Fanuc TP program (LS listing): DOOR_NOT_OP.LS

/PROG  DOOR_NOT_OP
/ATTR
OWNER		= MNEDITOR;
COMMENT		= "";
PROG_SIZE	= 170;
CREATE		= DATE 25-07-16  TIME 20:54:06;
MODIFIED	= DATE 25-07-16  TIME 20:54:40;
FILE_NAME	= ;
VERSION		= 0;
LINE_COUNT	= 2;
MEMORY_SIZE	= 542;
PROTECT		= READ_WRITE;
TCD:  STACK_SIZE	= 0,
      TASK_PRIORITY	= 50,
      TIME_SLICE	= 0,
      BUSY_LAMP_OFF	= 0,
      ABORT_REQUEST	= 0,
      PAUSE_REQUEST	= 0;
DEFAULT_GROUP	= *,*,*,*,*;
CONTROL_CODE	= 00000000 00000000;
/MN
   1:  UALM[2] ;
   2:  MONITOR DOOR_OP_COND ;
/POS
/END
